{attribute 'qualified_only'}
VAR_GLOBAL
	
	(*--------------- Omron TM5 Manipulator Parameters  ---------------*)
	{attribute 'OPC.UA.DA' := '1'}
	bStartTM	: BOOL;
	{attribute 'OPC.UA.DA' := '1'}
	bStopTM		: BOOL;
	
	
	{attribute 'OPC.UA.DA' := '1'}
	stRobotArmObjectTM : ST_RobotArmObjectTM;
	
	

	
	
	
	(*--------------- Omron LD-90 Mobile Robot Parameters  ---------------*)
	{attribute 'OPC.UA.DA' := '1'}
	bStartLD 	: BOOL;
	{attribute 'OPC.UA.DA' := '1'}
	bStopLD		: BOOL;
	statusReceivedLD 	: STRING(7680):= '';
	statusWriteLD 		: T_MaxString; 
	
	{attribute 'OPC.UA.DA' := '1'}
	stMobileRobotObjectLD : ST_MobileRobotObjectLD;

 

END_VAR

(* stored: Version 1.1.0.1, ProductVersion 3.1.4024.11
   GVL GVL_MobileManipulator: Id {d0a22671-0953-45c7-b5d6-9e717f6bd0a9} *)
